FUNCTION_BLOCK SET_AT_INDEX (* Service Interface Function Block Type *)
  (* Standard: 61499-2; Description: Set value of array at given index. Data types of value to be set must correspond to the array data type. Data type of resulting output array must correspond to input array data type. *)
  (* Version 0.0, 2014-07-11, Matthias Plasch, 4DIAC-Consortium *)
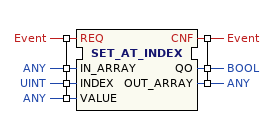
  EVENT_INPUT
    REQ WITH IN_ARRAY, INDEX, VALUE; (* Service Request *)
  END_EVENT
  EVENT_OUTPUT
    CNF WITH QO, OUT_ARRAY; (* Confirmation of Requested Service *)
  END_EVENT
  VAR_INPUT
    IN_ARRAY : ANY; (* input array *)
    INDEX : UINT; (* index to fetch value from *)
    VALUE : ANY; (* value to be copied to given index *)
  END_VAR
  VAR_OUTPUT
    QO : BOOL; (* Event Output Qualifier *)
    OUT_ARRAY : ANY; (* resulting array after set *)
  END_VAR
  (* Service APPLICATION/RESOURCE: Service Interface Function Block Type *)
END_FUNCTION_BLOCK
